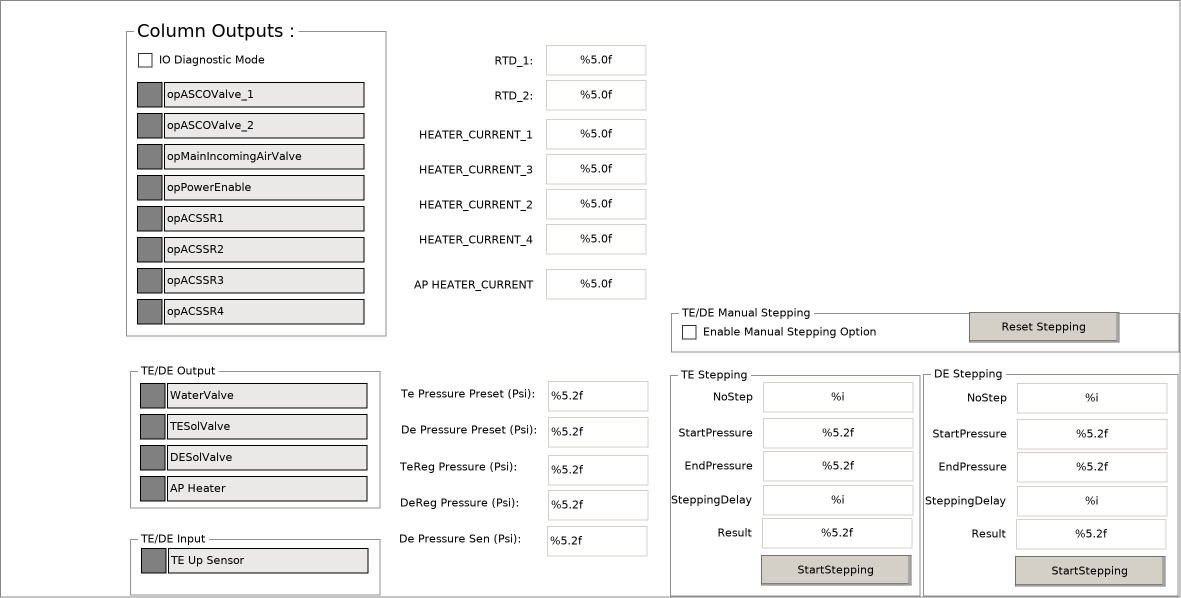
VISUALIZATION SLTC_Monitor  // 1181x598
    GroupBox (670,367 250x229), "TE Stepping"
    GroupBox (923,366 255x230), "DE Stepping"
    GroupBox (130,363 250x145), "TE/DE Output"
        RoundedRectangle (37,113 200x25), "AP Heater"
            toggle fbSLTCExtra.stDIO.opAPHeater
    GroupBox (130,531 250x64), "TE/DE Input"
    Textfield (546,45 100x30), "%5.0f", text variable: fbSLTCExtra.stVIO.ipRTD1
    Label (406,46 130x30), "RTD_1:"
    Textfield (546,80 100x30), "%5.0f", text variable: fbSLTCExtra.stVIO.ipRTD2
    Label (406,81 130x30), "RTD_2:"
    Textfield (546,119 100x30), "%5.0f", text variable: fbSLTCExtra.stVIO.ipHeaterCurrent1
    Label (406,120 130x30), "HEATER_CURRENT_1"
    Textfield (546,154 100x30), "%5.0f", text variable: fbSLTCExtra.stVIO.ipHeaterCurrent2
    Label (406,155 130x30), "HEATER_CURRENT_3"
    Textfield (546,189 100x30), "%5.0f", text variable: fbSLTCExtra.stVIO.ipHeaterCurrent3
    Label (406,190 130x30), "HEATER_CURRENT_2"
    Textfield (546,224 100x30), "%5.0f", text variable: fbSLTCExtra.stVIO.ipHeaterCurrent4
    Label (406,225 130x30), "HEATER_CURRENT_4"
    GroupBox (126,23 260x313), "Column Outputs :"
        RoundedRectangle (38,121 200x25), "opMainIncomingAirValve"
            toggle fbSLTCExtra.stDIO.opMainIncomingAirValve
        RoundedRectangle (38,183 200x25), "opACSSR1"
            toggle fbSLTCExtra.stDIO.opAC_SSR1
        RoundedRectangle (38,214 200x25), "opACSSR2"
            toggle fbSLTCExtra.stDIO.opAC_SSR2
        RoundedRectangle (11,121 25x25), colour toggle: fbSLTCExtra.stDIO.opMainIncomingAirValve
        RoundedRectangle (11,183 25x25), colour toggle: fbSLTCExtra.stDIO.opAC_SSR1
        RoundedRectangle (11,214 25x25), colour toggle: fbSLTCExtra.stDIO.opAC_SSR2
        RoundedRectangle (38,245 200x25), "opACSSR3"
            toggle fbSLTCExtra.stDIO.opAC_SSR3
        Checkbox (10,22 200x30), "IO Diagnostic Mode", variable: bColIODiagnosticsMode, invisible if: TRUE
    RoundedRectangle (164,82 200x25), "opASCOValve_1"
        toggle fbSLTCExtra.stDIO.opASCOValve_1
    RoundedRectangle (164,113 200x25), "opASCOValve_2"
        toggle fbSLTCExtra.stDIO.opASCOValve_2
    RoundedRectangle (137,82 25x25), colour toggle: fbSLTCExtra.stDIO.opASCOValve_1
    RoundedRectangle (137,113 25x25), colour toggle: fbSLTCExtra.stDIO.opASCOValve_2
    RoundedRectangle (164,299 200x25), "opACSSR4"
        toggle fbSLTCExtra.stDIO.opAC_SSR4
    RoundedRectangle (164,175 200x25), "opPowerEnable"
        toggle fbSLTCExtra.stDIO.opPowerEnable
    RoundedRectangle (137,268 25x25), colour toggle: fbSLTCExtra.stDIO.opAC_SSR3
    RoundedRectangle (137,299 25x25), colour toggle: fbSLTCExtra.stDIO.opAC_SSR4
    RoundedRectangle (137,175 25x25), colour toggle: fbSLTCExtra.stDIO.opPowerEnable
    RoundedRectangle (140,383 25x25), colour toggle: fbSLTCExtra.stDIO.opWaterValve
    RoundedRectangle (167,414 200x25), "TESolValve"
        toggle fbSLTCExtra.stDIO.opTESolValve
    RoundedRectangle (167,445 200x25), "DESolValve"
        toggle fbSLTCExtra.stDIO.opDESolValve
    RoundedRectangle (140,414 25x25), colour toggle: fbSLTCExtra.stDIO.opTESolValve
    RoundedRectangle (140,445 25x25), colour toggle: fbSLTCExtra.stDIO.opDESolValve
    RoundedRectangle (167,383 200x25), "WaterValve"
        toggle fbSLTCExtra.stDIO.opWaterValve
    RoundedRectangle (141,548 25x25), colour toggle: fbSLTCExtra.stDIO.ipTEUpRS
    RoundedRectangle (168,548 200x25), "TE Up Sensor"
    Textfield (548,381 100x30), "%5.2f", text variable: fbSLTCExtra.stVIO.opTEPressRegAOut, input disabled if: fbSLTCExtra.isEnManStepping
        OnMouseDown: write the text variable via Default, min 0, max 130
    Label (398,379 135x30), "Te Pressure Preset (Psi):"
    Textfield (548,417 100x30), "%5.2f", text variable: fbSLTCExtra.stVIO.opDEPressRegAOut
        OnMouseClick: write the text variable via Default, min 0, max 130
    Label (398,415 135x30), "De Pressure Preset (Psi):"
    Label (397,452 125x30), "TeReg Pressure (Psi):"
    Textfield (548,490 100x30), "%5.2f", text variable: fbSLTCExtra.stVIO.ipDEPressRegFeedBack
    Label (397,488 125x30), "DeReg Pressure (Psi):"
    Textfield (548,455 100x30), "%5.2f", text variable: fbSLTCExtra.stVIO.ipTEPressRegFeedBack
    Textfield (547,526 100x30), "%5.2f", text variable: fbSLTCExtra.stVIO.ipDEPressureSensor
    Label (396,524 125x30), "De Pressure Sen (Psi):"
    Textfield (763,382 150x30), "%i", text variable: fbSLTCExtra.noOfStepTE, input disabled if: Not fbSLTCExtra.isEnManStepping
        OnMouseClick: write the text variable via Default
    Label (666,382 90x30), "NoStep"
    Button (761,555 150x30), "StartStepping", input disabled if: fbSLTCExtra.isStartSteppingTE OR Not fbSLTCExtra.isEnManStepping
        tap fbSLTCExtra.btnToggleTE p1329445385=TRUE
    Textfield (763,418 150x30), "%5.2f", text variable: fbSLTCExtra.startPressureTE, input disabled if: Not fbSLTCExtra.isEnManStepping
        OnMouseClick: write the text variable via Default
    Label (666,418 90x30), "StartPressure"
    Textfield (763,451 150x30), "%5.2f", text variable: fbSLTCExtra.endPressureTE, input disabled if: Not fbSLTCExtra.isEnManStepping
        OnMouseClick: write the text variable via Default
    Label (666,451 90x30), "EndPressure"
    Textfield (763,485 150x30), "%i", text variable: fbSLTCExtra.StepDelayTE, input disabled if: Not fbSLTCExtra.isEnManStepping
        OnMouseClick: write the text variable via Default
    Label (665,485 90x30), "SteppingDelay"
    Label (665,518 90x30), "Result"
    Textfield (762,518 150x30), "%5.2f", text variable: fbSLTCExtra.TEResult, input disabled if: TRUE
    Checkbox (680,317 215x30), "Enable Manual Stepping Option", variable: fbSLTCExtra.isEnManStepping
    Textfield (1017,383 150x30), "%i", text variable: fbSLTCExtra.noOfStepDE, input disabled if: Not fbSLTCExtra.isEnManStepping
        OnMouseClick: write the text variable via Default
    Label (920,383 90x30), "NoStep"
    Button (1015,556 150x30), "StartStepping", input disabled if: fbSLTCExtra.isStartSteppingDE OR Not fbSLTCExtra.isEnManStepping
        tap fbSLTCExtra.btnToggleDE p1329445385=TRUE
    Textfield (1017,419 150x30), "%5.2f", text variable: fbSLTCExtra.startPressureDE, input disabled if: Not fbSLTCExtra.isEnManStepping
        OnMouseClick: write the text variable via Default
    Label (920,419 90x30), "StartPressure"
    Textfield (1017,452 150x30), "%5.2f", text variable: fbSLTCExtra.endPressureDE, input disabled if: Not fbSLTCExtra.isEnManStepping
        OnMouseClick: write the text variable via Default
    Label (920,452 90x30), "EndPressure"
    Textfield (1017,486 150x30), "%i", text variable: fbSLTCExtra.StepDelayDE, input disabled if: Not fbSLTCExtra.isEnManStepping
        OnMouseClick: write the text variable via Default
    Label (919,486 90x30), "SteppingDelay"
    Label (919,519 90x30), "Result"
    Textfield (1016,519 150x30), "%5.2f", text variable: fbSLTCExtra.DEResult, input disabled if: TRUE
    GroupBox (671,305 508x47), "TE/DE Manual Stepping"
        Button (298,7 150x30), "Reset Stepping", input disabled if: fbSLTCExtra.isStartSteppingTE AND fbSLTCExtra.isStartSteppingDE OR Not fbSLTCExtra.isEnManStepping
            tap fbSLTCExtra.isResetStepping
    RoundedRectangle (140,476 25x25), colour toggle: fbSLTCExtra.stDIO.opAPHeater
    Textfield (546,269 100x30), "%5.0f", text variable: fbSLTCExtra.stVIO.ipAPHeaterCurrent
    Label (388,270 148x30), "AP HEATER_CURRENT"
END_VISUALIZATION

(* stored: Version 1.1.0.1, ProductVersion 3.1.4022.12
   Visu SLTC_Monitor: Id {1adf1e04-6bce-4280-9cf1-0162170a5674} *)
